// TIA Portal V20 export
// export: Created 2026-08-20T19:00:41.1350475Z, ExportSetting WithDefaults, DisplayName Totally Integrated Automation Portal, DisplayVersion V20, DisplayName TIA Portal Openness, DisplayVersion V20, DisplayName TIA Portal Version Control Interface, DisplayVersion V20, DisplayName STEP 7 Professional, DisplayVersion V20, DisplayName STEP 7 Safety, DisplayVersion V20, DisplayName WinCC Basic/Comfort/Advanced, DisplayVersion V20, DisplayName WinCC Unified, DisplayVersion V20
ORGANIZATION_BLOCK "Main"   // OB1, LAD, ProgramCycle
TITLE = "Main Program Sweep (Cycle)"
{ S7_Optimized_Access := 'TRUE' }
VERSION : 0.1
// stored: AutoNumber true, IsIECCheckEnabled false, SetENOAutomatically false
   VAR_INPUT
      Initial_Call : Bool;   // Initial call of this OB
      Remanence : Bool;   // =True, if remanent data are available
   END_VAR
BEGIN

REGION Network 1
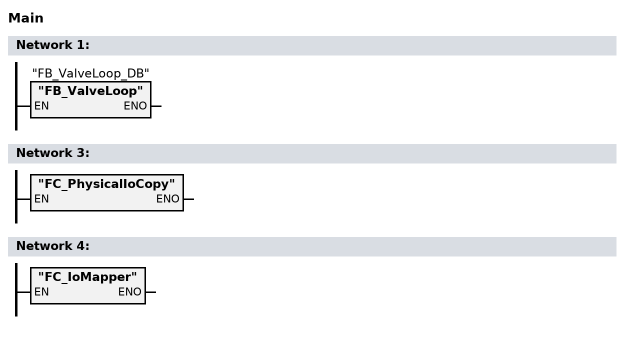
   RUNG wire#powerrail
      "FB_ValveLoop_DB"()
   END_RUNG
   // the same network as SCL:
   "FB_ValveLoop_DB"();   // "FB_ValveLoop"
END_REGION

REGION Network 3
   RUNG wire#powerrail
      "FC_PhysicalIoCopy"()
   END_RUNG
   // the same network as SCL:
   "FC_PhysicalIoCopy"();
END_REGION

REGION Network 4
   RUNG wire#powerrail
      "FC_IoMapper"()
   END_RUNG
   // the same network as SCL:
   "FC_IoMapper"();
END_REGION
END_ORGANIZATION_BLOCK
